(* PLC project codesysFlow11plus.project, CODESYS CODESYS V3.5 SP17 Patch 3 *)
(* stored: creationDateTime 2022-12-19T23:42:12.4738087, modificationDateTime 2022-12-18T10:15:13.8942381 *)

PROGRAM POU2_1
  VAR
    t0 : BOOL;
    t1 : BOOL;
    t2 : BOOL;
    t3 : BOOL;
    t4 : BOOL;
    t5 : BOOL;
    t6 : BOOL;
    t7 : BOOL;
    t8 : BOOL;
    t9 : BOOL;
    t10 : BOOL;
    t11 : BOOL;
    t12 : BOOL;
    t13 : BOOL;
    t14 : BOOL;
    t15 : BOOL;
    t16 : BOOL;
    t17 : BOOL;
    t18 : BOOL;
    t19 : BOOL;
    t20 : BOOL;
    t21 : BOOL;
    t22 : BOOL;
    t23 : BOOL;
    t24 : BOOL;
    t25 : BOOL;
    t26 : BOOL;
    t27 : BOOL;
    t28 : BOOL;
    t29 : BOOL;
  END_VAR

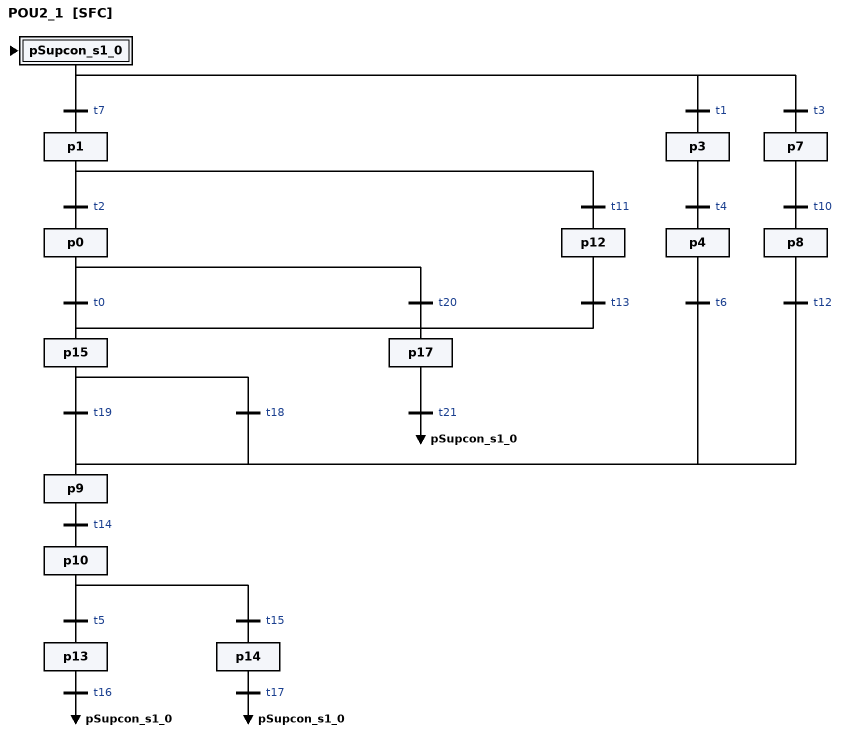
INITIAL_STEP pSupcon_s1_0:
END_STEP
TRANSITION FROM pSupcon_s1_0 TO p1
  := t7;
END_TRANSITION
TRANSITION FROM pSupcon_s1_0 TO p3
  := t1;
END_TRANSITION
TRANSITION FROM pSupcon_s1_0 TO p7
  := t3;
END_TRANSITION
STEP p1:
END_STEP
TRANSITION FROM p1 TO p0
  := t2;
END_TRANSITION
TRANSITION FROM p1 TO p12
  := t11;
END_TRANSITION
STEP p0:
END_STEP
TRANSITION FROM p0 TO p15
  := t0;
END_TRANSITION
TRANSITION FROM p0 TO p17
  := t20;
END_TRANSITION
STEP p17:
END_STEP
TRANSITION FROM p17 TO pSupcon_s1_0
  := t21;
END_TRANSITION
STEP p12:
END_STEP
TRANSITION FROM p12 TO p15
  := t13;
END_TRANSITION
STEP p15:
END_STEP
TRANSITION FROM p15 TO p9
  := t19;
END_TRANSITION
TRANSITION FROM p15 TO p9
  := t18;
END_TRANSITION
STEP p3:
END_STEP
TRANSITION FROM p3 TO p4
  := t4;
END_TRANSITION
STEP p4:
END_STEP
TRANSITION FROM p4 TO p9
  := t6;
END_TRANSITION
STEP p7:
END_STEP
TRANSITION FROM p7 TO p8
  := t10;
END_TRANSITION
STEP p8:
END_STEP
TRANSITION FROM p8 TO p9
  := t12;
END_TRANSITION
STEP p9:
END_STEP
TRANSITION FROM p9 TO p10
  := t14;
END_TRANSITION
STEP p10:
END_STEP
TRANSITION FROM p10 TO p13
  := t5;
END_TRANSITION
TRANSITION FROM p10 TO p14
  := t15;
END_TRANSITION
STEP p13:
END_STEP
TRANSITION FROM p13 TO pSupcon_s1_0
  := t16;
END_TRANSITION
STEP p14:
END_STEP
TRANSITION FROM p14 TO pSupcon_s1_0
  := t17;
END_TRANSITION
END_PROGRAM
